SUBAPPLICATION Uebung_070c (* WBSD auf UT ausgeben, PHYS *)
  (* Standard: 61499-2; Description: Copyright (c) 2023 Meisterschulen am Ostbahnhof This program and the accompanying materials are made available under the terms of the Eclipse Public License 2.0 which is available at https://www.eclipse.org/legal/epl-2.0/ SPDX-License-Identifier: EPL-2.0 *)
  (* Version 1.0, 2023-10-23, Franz Höpfinger, Meisterschulen am Ostbahnhof, initial API and implementation and/or initial documentation *)
  PACKAGE Uebungen;
  IMPORT Uebungen::const::UT::TECU::DefaultPool_TECU_Numeric::NumberVariable_Wheel_based_machine_speed_N;
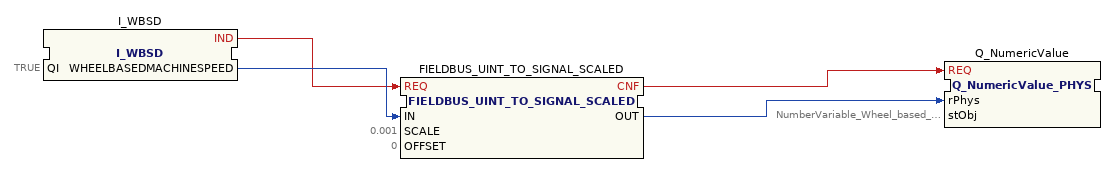
  FBS
    I_WBSD : isobus::tecu::I_WBSD(QI := TRUE);
    Q_NumericValue : isobus::UT::Q::Q_NumericValue_PHYS(stObj := NumberVariable_Wheel_based_machine_speed_N);
    FIELDBUS_UINT_TO_SIGNAL_SCALED : logiBUS::signalprocessing::fieldbus::FIELDBUS_UINT_TO_SIGNAL_SCALED(SCALE := 0.001, OFFSET := 0);
  END_FBS
  EVENT_CONNECTIONS
    I_WBSD.IND TO FIELDBUS_UINT_TO_SIGNAL_SCALED.REQ;
    FIELDBUS_UINT_TO_SIGNAL_SCALED.CNF TO Q_NumericValue.REQ;
  END_CONNECTIONS
  DATA_CONNECTIONS
    I_WBSD.WHEELBASEDMACHINESPEED TO FIELDBUS_UINT_TO_SIGNAL_SCALED.IN;
    FIELDBUS_UINT_TO_SIGNAL_SCALED.OUT TO Q_NumericValue.rPhys;
  END_CONNECTIONS
END_SUBAPPLICATION
